{attribute 'qualified_only'}
VAR_GLOBAL CONSTANT
	tSamplePeriodic : TIME := T#30S; // Interval of sample periodic meter values in FB_ConnectorMeter
	tSampleClock : TIME := T#60S; // Interval of sample clock meter values in FB_StationMeter
END_VAR

(* stored: Version 1.1.0.1
   GVL VAR_Param: Id {4877451f-5147-4895-8ce1-fddd84565e5e} *)
